PROGRAM systime
VAR
	fb_localsystime1:Tc2_Utilities.FB_LocalSystemTime;
	systime1:Tc2_Utilities.TIMESTRUCT;
	dttime:DATE_AND_TIME;
	todacttime:TIME_OF_DAY;
	sTime,sData	:STRING;
END_VAR

fb_localsystime1(
	sNetID:= , 
	bEnable:= TRUE, 
	dwCycle:= , 
	dwOpt:= , 
	tTimeout:= , 
	bValid=> , 
	systemTime=>systime1 , 
	tzID=> );
	
dttime:=Tc2_Utilities.SYSTEMTIME_TO_DT(systime1);
todacttime:=DT_TO_TOD(dttime);
    sTime := concat(WORD_TO_STRING(fb_localsystime1.systemTime.wHour),':');
	sTime := concat(sTime,WORD_TO_STRING(fb_localsystime1.systemTime.wMinute));
	sTime := concat(sTime,':');
	sTime := concat(sTime,WORD_TO_STRING(fb_localsystime1.systemTime.wSecond));
(*	sData := concat(WORD_TO_STRING(fb_localsystime1.systemTime.wDayOfWeek),',');
	sData := Tc2_Standard.CONCAT(sData,WORD_TO_STRING(fb_localsystime1.systemTime.wMonth));
	sData := Tc2_Standard.CONCAT(sdata,'.');
	sData := Tc2_Standard.CONCAT(sData,WORD_TO_STRING(fb_localsystime1.systemTime.wDay));
	sData := Tc2_Standard.CONCAT(sData,',');
	sData := Tc2_Standard.CONCAT(sData,WORD_TO_STRING(fb_localsystime1.systemTime.wYear));
	*)

END_PROGRAM

(* stored: Version 1.1.0.1, ProductVersion 3.1.4024.11
   POU systime: Id {ae3e90b9-ad75-49d9-b5f3-1b0198564b79}, SpecialFunc None *)
